(* CODESYS project semaforoV35V11.project

Project tree, tasks and I/O mapping:
  CODESYS_Control_Win_V3 : CODESYS Control Win V3, 3S - Smart Software Solutions GmbH, order no. 305021, version 3.5.11.30
    application Application
      libraries: Standard, * (System)
      task VISU_TASK (cyclic, interval 100 ms, priority 31) calls VisuElems.Visu_Prg, PLC_PRG
      program PLC_PRG [ST]
      visualisation Visualization
  libraries: VisuSymbols, 3.5.10.0 (System)
  text list GlobalTextList
*)

// CODESYS_Control_Win_V3/Application/PLC_PRG
PROGRAM PLC_PRG
VAR
	B1:BOOL; // Botão de Inicialização
	P0:BOOL; // Passo inicial
	P1:BOOL; // Passo 1
	P2:BOOL; // Passo 2
	P3:BOOL; // Passo 3
	P4:BOOL; // Passo 4
	P5:BOOL; // Passo 5
	PULSOS_OUT_1: BOOL; // Variável de saída do gerador de pulsos
	PULSOS_OUT_2: BOOL; // Variável de saída do gerador de pulsos
	ET1:TIME; // Variável de tempo do timer 1
	ET2:TIME; // Variável de tempo do timer 2
	ET3:TIME; // Variável de tempo do timer 3
	ET4:TIME; // Variável de tempo do timer 4
	ET5:TIME; // Variável de tempo do timer 5
	ET_PULSOS_1: TIME; // Variável de pulsos
	ET_PULSOS_2: TIME; // Variável de pulsos
	S1_V: BOOL; // Luz verde do semáforo 1
	S1_A: BOOL; // Luz amarela do semáforo 1
	S1_M: BOOL; // Luz vermelha do semáforo 1
	S2_V: BOOL; // Luz verde do semáforo 2
	S2_A: BOOL; // Luz amarela do semáforo 2
	S2_M: BOOL; // Luz vermelha do semáforo 2
	S3_V: BOOL; // Luz verde do semáforo 3
	S3_A: BOOL; // Luz amarela do semáforo 3
	S3_M: BOOL; // Luz vermelha do semáforo 3
	S3_AZUL: BOOL; // Luz azul do semáforo 3
	RT0: R_TRIG; // Rasing trigger 0
	FT1: F_TRIG; // Falling trigger 1
	FT2: F_TRIG; // Falling trigger 2
	FT3: F_TRIG; // Falling trigger 3
	FT4: F_TRIG; // Falling trigger 4
	FT5: F_TRIG; // Falling trigger 5
	FT_PULSOS_1: F_TRIG; // Função falling trigger 1
	FT_PULSOS_2: F_TRIG; // Função falling trigger 2
	FT_PULSOS_3: F_TRIG; // Função falling trigger 3
    T1:TP; // Timer de Pulso 1
    T2:TP; // Timer de Pulso 2
    T3:TP; // Timer de Pulso 3
    T4:TP; // Timer de Pulso 4
    T5:TP; // Timer de Pulso 5
	TP_PULSOS_1: TP; // Timer de pulsos 1
	TP_PULSOS_2: TP; // Timer de pulsos 2
END_VAR


FT_PULSOS_1(CLK:=B1); // Se o botão gerar uma transição de 1 para 0 aciona a saída do FT_PULSOS1
IF (B1 = FALSE) THEN //Verifica se o botão está em nível lógico 0
	TP_PULSOS_1(IN:=(FT_PULSOS_1.Q OR FT_PULSOS_3.Q),PT:=T#1S,ET=>ET_PULSOS_1,Q=>PULSOS_OUT_1); 
	FT_PULSOS_2(CLK:=PULSOS_OUT_1);
	TP_PULSOS_2(IN:=FT_PULSOS_2.Q,PT:=T#1S,ET=>ET_PULSOS_2,Q=>PULSOS_OUT_2); 
	FT_PULSOS_3(CLK:=PULSOS_OUT_2);
	
	S1_V:= FALSE;
	S1_A:= PULSOS_OUT_1;
	S1_M:= FALSE;
    S2_V:= FALSE;
	S2_A:= PULSOS_OUT_1;
	S2_M:= FALSE;
    S3_V:= FALSE;
	S3_A:= PULSOS_OUT_1;
	S3_M:= FALSE;
	S3_AZUL := FALSE;
END_IF



P0 := B1; // Passo 0 acionado pelo botão B1
RT0(CLK:=P0); // Função rasing trigger acionada pelo passo P0

IF (B1 = TRUE) THEN //Verifica se o botão está em nível lógico 1
	T1(IN:=(RT0.Q OR FT5.Q),PT:=T#15S,ET=>ET1,Q=>P1); // Timer de pulso 1 acionado pela função RT0 ou FT5 (fecha o ciclo)

	FT1(CLK:=P1); // Função FT1 (falling trigger) acionada pelo passo P1
	T2(IN:=FT1.Q,PT:=T#5S,ET=>ET2,Q=>P2);  // Timer de pulso 2 acionado pela função FT1 falling trigger)

	FT2(CLK:=P2); // Função FT2 (falling trigger) acionada pelo passo P2
	T3(IN:=FT2.Q,PT:=T#15S,ET=>ET3,Q=>P3); // Timer de pulso 3 acionado pela função FT2 (falling trigger)

	FT3(CLK:=P3); // Função FT3 (falling trigger) acionada pelo passo P3
	T4(IN:=FT3.Q,PT:=T#5S,ET=>ET4,Q=>P4); // Timer de pulso 4 acionado pela função FT3 (falling trigger)

	FT4(CLK:=P4); // Função FT4 (falling trigger) acionada pelo passo P4
	T5(IN:=FT4.Q,PT:=T#10S,ET=>ET5,Q=>P5); // Timer de pulso 5 acionado pela função FT4 (falling trigger)

	FT5(CLK:=P5); // Função FT5 (falling trigger) acionada pelo passo P5

	IF (P1 = TRUE) THEN // Se o passo P1 for TRUE acender as seguintes luzes
		S1_V:= TRUE;
		S1_A:= FALSE;
		S1_M:= FALSE;
    	S2_V:= FALSE;
		S2_A:= FALSE;
		S2_M:= TRUE;
    	S3_V:= FALSE;
		S3_A:= FALSE;
		S3_M:= TRUE;
		S3_AZUL := FALSE;
	ELSIF (P2 = TRUE) THEN // Se o passo P2 for TRUE acender as seguintes luzes
		S1_V:= FALSE;
		S1_A:= TRUE;
		S1_M:= FALSE;
    	S2_V:= FALSE;
		S2_A:= FALSE;
		S2_M:= TRUE;
    	S3_V:= FALSE;
		S3_A:= FALSE;
		S3_M:= TRUE;
		S3_AZUL := FALSE;
	ELSIF (P3 = TRUE) THEN // Se o passo P3 for TRUE acender as seguintes luzes
		S1_V:= FALSE;
		S1_A:= FALSE;
		S1_M:= TRUE;
    	S2_V:= TRUE;
		S2_A:= FALSE;
		S2_M:= FALSE;
    	S3_V:= TRUE;
		S3_A:= FALSE;
		S3_M:= FALSE;
		S3_AZUL := FALSE;
	ELSIF (P4 = TRUE) THEN // Se o passo P4 for TRUE acender as seguintes luzes
		S1_V:= FALSE;
		S1_A:= FALSE;
		S1_M:= TRUE;
    	S2_V:= FALSE;
		S2_A:= TRUE;
		S2_M:= FALSE;
    	S3_V:= TRUE;
		S3_A:= FALSE;
		S3_M:= FALSE;
		S3_AZUL := FALSE;
	ELSIF (P5 = TRUE) THEN // Se o passo P5 for TRUE acender as seguintes luzes
		S1_V:= FALSE;
		S1_A:= FALSE;
		S1_M:= TRUE;
    	S2_V:= FALSE;
		S2_A:= FALSE;
		S2_M:= TRUE;
    	S3_V:= FALSE;
		S3_A:= FALSE;
		S3_M:= FALSE;
		S3_AZUL := TRUE;
	END_IF

END_IF

END_PROGRAM

// CODESYS_Control_Win_V3/Application/Visualization
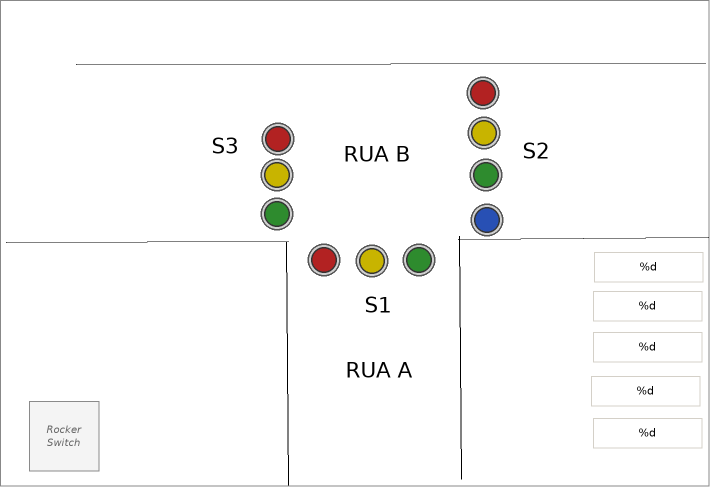
VISUALIZATION Visualization  // 710x487
    Lamp1 (305,239 38x42), variable: PLC_PRG.S1_M, style: Lamp-Lamp1-Red
    RockerSwitch (29,401 70x70), variable: PLC_PRG.B1, behaviour: TOGGLE, style: Switch-RockerSwitch-Gray
    Line (76,64) (705,63)
    Line (6,242) (288,241)
    Line (458,239) (708,237)
    Line (286,242) (288,485)
    Line (459,236) (461,479)
    Lamp1 (353,240 38x42), variable: PLC_PRG.S1_A, style: Lamp-Lamp1-Yellow
    Lamp1 (400,239 38x42), variable: PLC_PRG.S1_V, style: Lamp-Lamp1-Green
    Lamp1 (259,118 38x42), variable: PLC_PRG.S2_M, style: Lamp-Lamp1-Red
    Lamp1 (258,154 38x42), variable: PLC_PRG.S2_A, style: Lamp-Lamp1-Yellow
    Lamp1 (258,193 38x42), variable: PLC_PRG.S2_V, style: Lamp-Lamp1-Green
    Lamp1 (464,72 38x42), variable: PLC_PRG.S3_M, style: Lamp-Lamp1-Red
    Lamp1 (465,112 38x42), variable: PLC_PRG.S3_A, style: Lamp-Lamp1-Yellow
    Lamp1 (467,154 38x42), variable: PLC_PRG.S3_V, style: Lamp-Lamp1-Green
    Lamp1 (468,199 38x42), variable: PLC_PRG.S3_AZUL, style: Lamp-Lamp1-Blue
    Textfield (594,252 109x30), "%d", text variable: PLC_PRG.ET1
    Textfield (593,291 109x30), "%d", text variable: PLC_PRG.ET2
    Textfield (593,332 109x30), "%d", text variable: PLC_PRG.ET3
    Textfield (591,376 109x30), "%d", text variable: PLC_PRG.ET4
    Textfield (593,418 109x30), "%d", text variable: PLC_PRG.ET5
    Label (328,139 98x30), "RUA B"
    Label (330,355 98x30), "RUA A"
    Label (329,290 98x30), "S1"
    Label (487,136 98x30), "S2"
    Label (176,131 98x30), "S3"
END_VISUALIZATION
